Fanuc KAREL source: ko00028.KL

-- PROVISIONAL review KL for V940-1; original PC SHA256 e859606e251a0f5954eba6bf828e218edbd6af2f1a85ad14bd34f1d07abd6c99
-- Incomplete behavior may be omitted. Consult companion uncertainty JSON. Do not deploy.
PROGRAM KO00028
%NOLOCKGROUP
-- UNRESOLVED_DECL P1 type=000199
-- UNRESOLVED_DECL P2 type=000199
-- UNRESOLVED_DECL P3 type=000199
-- UNRESOLVED_DECL OUT type=000199
BEGIN
  -- V9_ZERO_TABLE_METADATA_HINT layout=0001; no indexed target words; source/name/runtime held
  -- UNRESOLVED_PC offsets 5-65; opcodes 27,27,49,7E,AD,27,49,7E,AD,27,49,7E,AD,76,7E,4A
  -- UNRESOLVED_PC offsets 70-74; opcodes 7F
END KO00028
